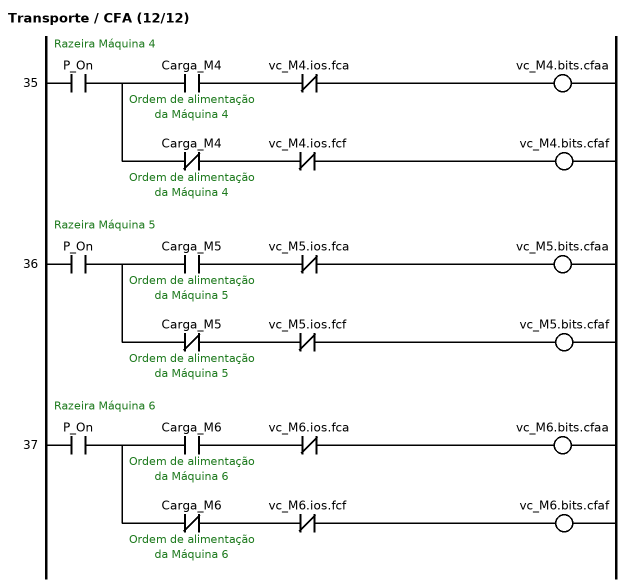
; [picture p24: Transporte / CFA, rungs 35-37]
; rung 35: Razeira Máquina 4
LD P_On
OUT TR0
AND Carga_M4  ; Ordem de alimentação da Máquina 4
ANDNOT vc_M4.ios.fca
OUT vc_M4.bits.cfaa
LD TR0
ANDNOT Carga_M4  ; Ordem de alimentação da Máquina 4
ANDNOT vc_M4.ios.fcf
OUT vc_M4.bits.cfaf
; rung 36: Razeira Máquina 5
LD P_On
OUT TR0
AND Carga_M5  ; Ordem de alimentação da Máquina 5
ANDNOT vc_M5.ios.fca
OUT vc_M5.bits.cfaa
LD TR0
ANDNOT Carga_M5  ; Ordem de alimentação da Máquina 5
ANDNOT vc_M5.ios.fcf
OUT vc_M5.bits.cfaf
; rung 37: Razeira Máquina 6
LD P_On
OUT TR0
AND Carga_M6  ; Ordem de alimentação da Máquina 6
ANDNOT vc_M6.ios.fca
OUT vc_M6.bits.cfaa
LD TR0
ANDNOT Carga_M6  ; Ordem de alimentação da Máquina 6
ANDNOT vc_M6.ios.fcf
OUT vc_M6.bits.cfaf

### Section FCOMUNICACAO

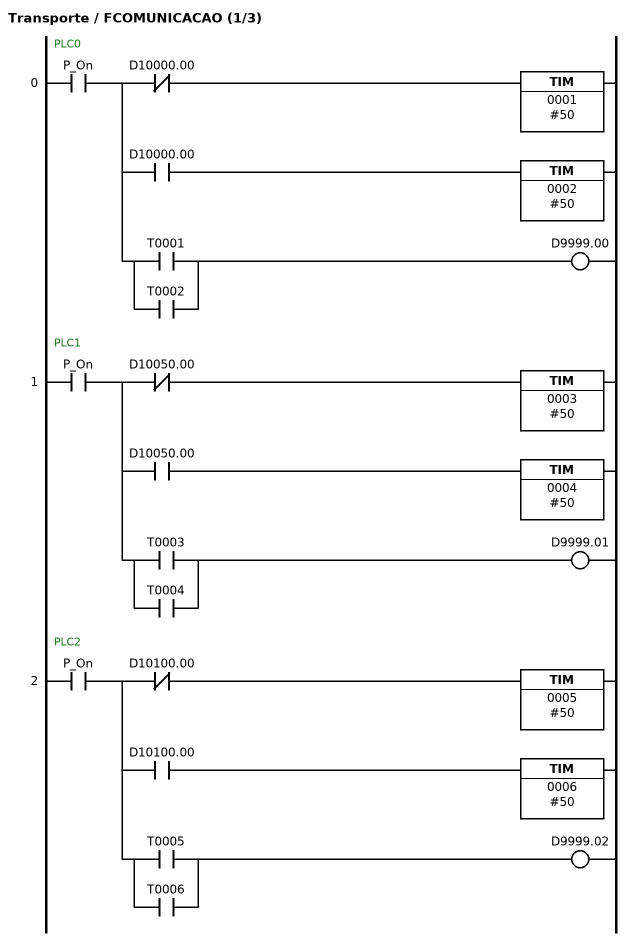
; rung 0: PLC0
LD P_On
OUT TR0
ANDNOT D10000.00
TIM 0001 #50
LD TR0
AND D10000.00
TIM 0002 #50
LD TR0
LD T0001
OR T0002
ANDLD
OUT D9999.00
; rung 1: PLC1
LD P_On
OUT TR0
ANDNOT D10050.00
TIM 0003 #50
LD TR0
AND D10050.00
TIM 0004 #50
LD TR0
LD T0003
OR T0004
ANDLD
OUT D9999.01
; rung 2: PLC2
LD P_On
OUT TR0
ANDNOT D10100.00
TIM 0005 #50
LD TR0
AND D10100.00
TIM 0006 #50
LD TR0
LD T0005
OR T0006
ANDLD
OUT D9999.02

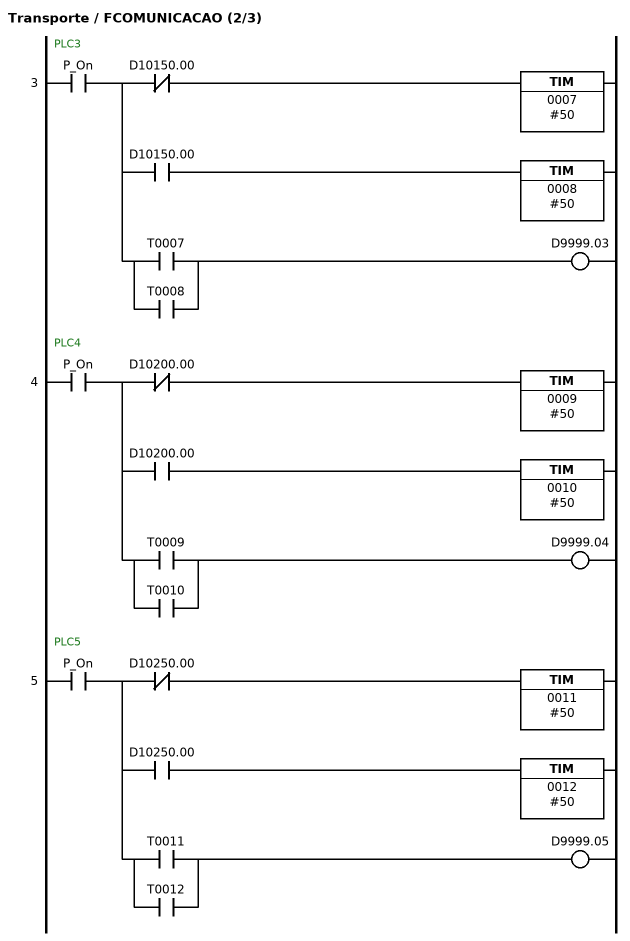
; rung 3: PLC3
LD P_On
OUT TR0
ANDNOT D10150.00
TIM 0007 #50
LD TR0
AND D10150.00
TIM 0008 #50
LD TR0
LD T0007
OR T0008
ANDLD
OUT D9999.03
; rung 4: PLC4
LD P_On
OUT TR0
ANDNOT D10200.00
TIM 0009 #50
LD TR0
AND D10200.00
TIM 0010 #50
LD TR0
LD T0009
OR T0010
ANDLD
OUT D9999.04
; rung 5: PLC5
LD P_On
OUT TR0
ANDNOT D10250.00
TIM 0011 #50
LD TR0
AND D10250.00
TIM 0012 #50
LD TR0
LD T0011
OR T0012
ANDLD
OUT D9999.05

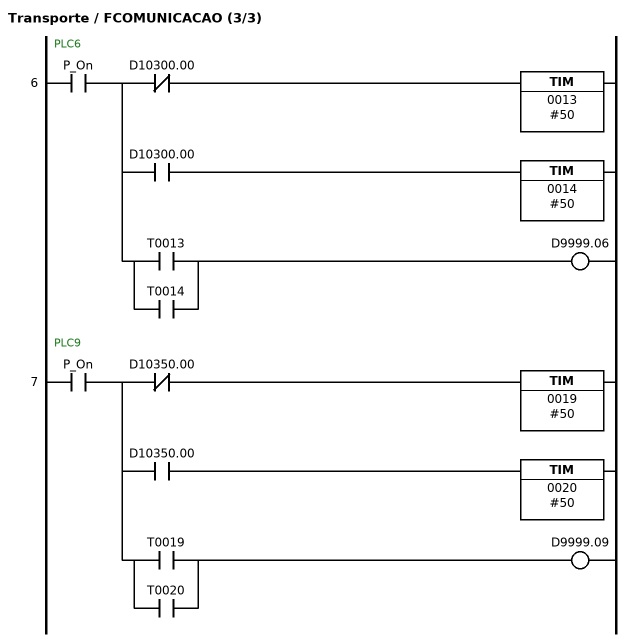
; rung 6: PLC6
LD P_On
OUT TR0
ANDNOT D10300.00
TIM 0013 #50
LD TR0
AND D10300.00
TIM 0014 #50
LD TR0
LD T0013
OR T0014
ANDLD
OUT D9999.06
; rung 7: PLC9
LD P_On
OUT TR0
ANDNOT D10350.00
TIM 0019 #50
LD TR0
AND D10350.00
TIM 0020 #50
LD TR0
LD T0019
OR T0020
ANDLD
OUT D9999.09

### Section COMUNICACAO

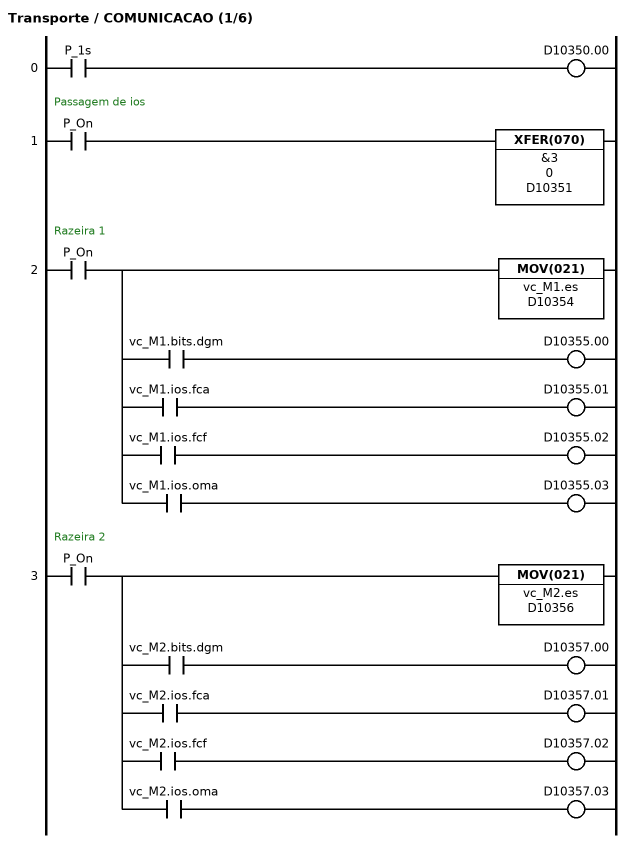
; rung 0
LD P_1s
OUT D10350.00
; rung 1: Passagem de ios
LD P_On
XFER(070) &3 0 D10351
; rung 2: Razeira 1
LD P_On
OUT TR0
MOV(021) vc_M1.es D10354
AND vc_M1.bits.dgm
OUT D10355.00
LD TR0
AND vc_M1.ios.fca
OUT D10355.01
LD TR0
AND vc_M1.ios.fcf
OUT D10355.02
LD TR0
AND vc_M1.ios.oma
OUT D10355.03
; rung 3: Razeira 2
LD P_On
OUT TR0
MOV(021) vc_M2.es D10356
AND vc_M2.bits.dgm
OUT D10357.00
LD TR0
AND vc_M2.ios.fca
OUT D10357.01
LD TR0
AND vc_M2.ios.fcf
OUT D10357.02
LD TR0
AND vc_M2.ios.oma
OUT D10357.03

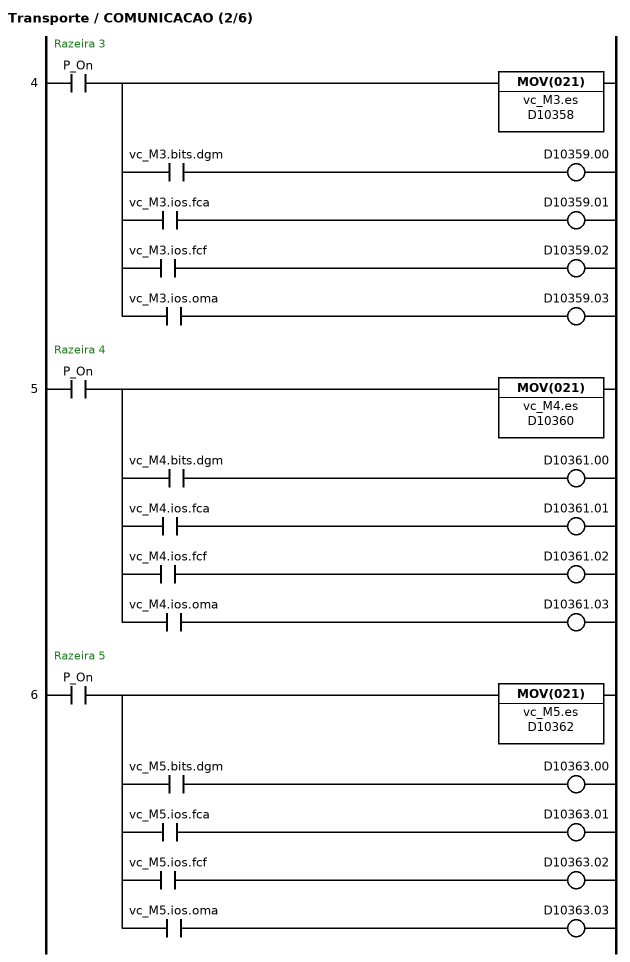
; rung 4: Razeira 3
LD P_On
OUT TR0
MOV(021) vc_M3.es D10358
AND vc_M3.bits.dgm
OUT D10359.00
LD TR0
AND vc_M3.ios.fca
OUT D10359.01
LD TR0
AND vc_M3.ios.fcf
OUT D10359.02
LD TR0
AND vc_M3.ios.oma
OUT D10359.03
; rung 5: Razeira 4
LD P_On
OUT TR0
MOV(021) vc_M4.es D10360
AND vc_M4.bits.dgm
OUT D10361.00
LD TR0
AND vc_M4.ios.fca
OUT D10361.01
LD TR0
AND vc_M4.ios.fcf
OUT D10361.02
LD TR0
AND vc_M4.ios.oma
OUT D10361.03
; rung 6: Razeira 5
LD P_On
OUT TR0
MOV(021) vc_M5.es D10362
AND vc_M5.bits.dgm
OUT D10363.00
LD TR0
AND vc_M5.ios.fca
OUT D10363.01
LD TR0
AND vc_M5.ios.fcf
OUT D10363.02
LD TR0
AND vc_M5.ios.oma
OUT D10363.03

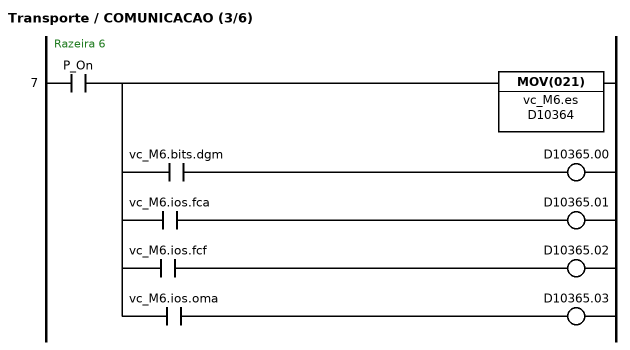
; rung 7: Razeira 6
LD P_On
OUT TR0
MOV(021) vc_M6.es D10364
AND vc_M6.bits.dgm
OUT D10365.00
LD TR0
AND vc_M6.ios.fca
OUT D10365.01
LD TR0
AND vc_M6.ios.fcf
OUT D10365.02
LD TR0
AND vc_M6.ios.oma
OUT D10365.03

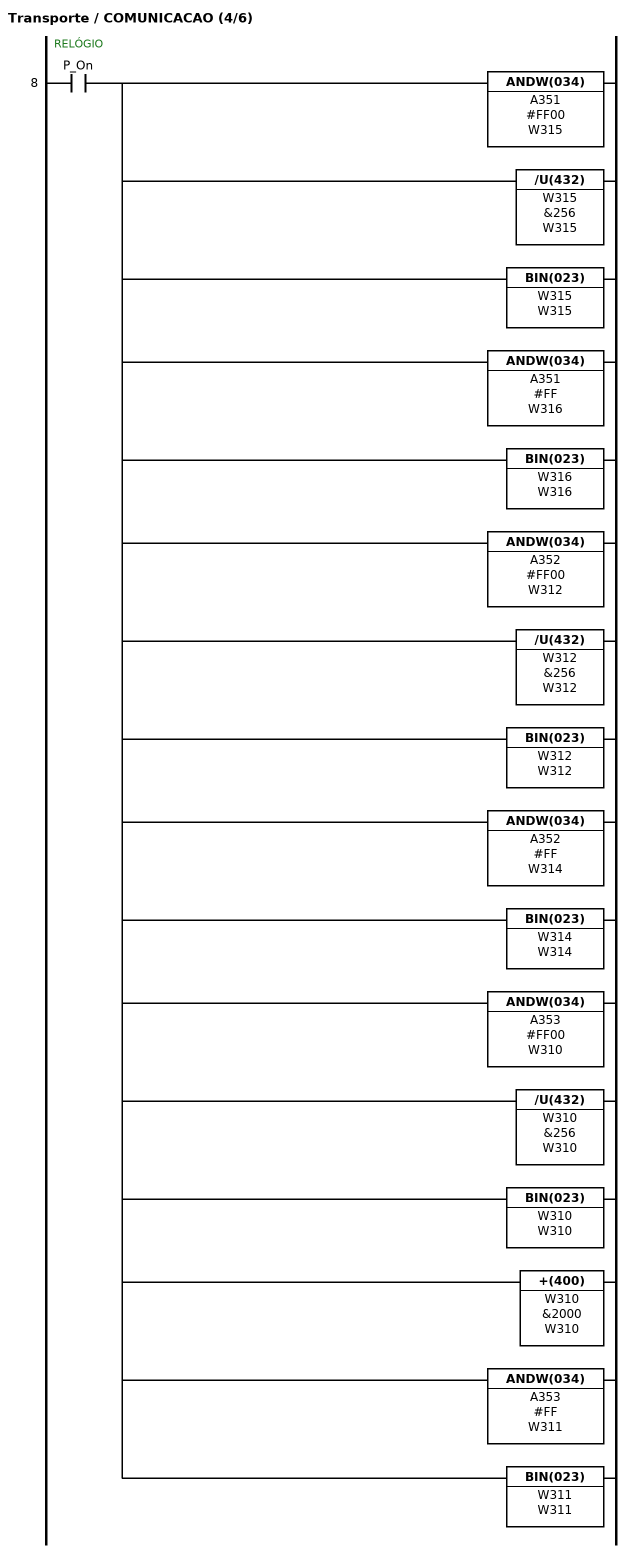
; rung 8: RELÓGIO
LD P_On
ANDW(034) A351 #FF00 W315
/U(432) W315 &256 W315
BIN(023) W315 W315
ANDW(034) A351 #FF W316
BIN(023) W316 W316
ANDW(034) A352 #FF00 W312
/U(432) W312 &256 W312
BIN(023) W312 W312
ANDW(034) A352 #FF W314
BIN(023) W314 W314
ANDW(034) A353 #FF00 W310
/U(432) W310 &256 W310
BIN(023) W310 W310
+(400) W310 &2000 W310
ANDW(034) A353 #FF W311
BIN(023) W311 W311

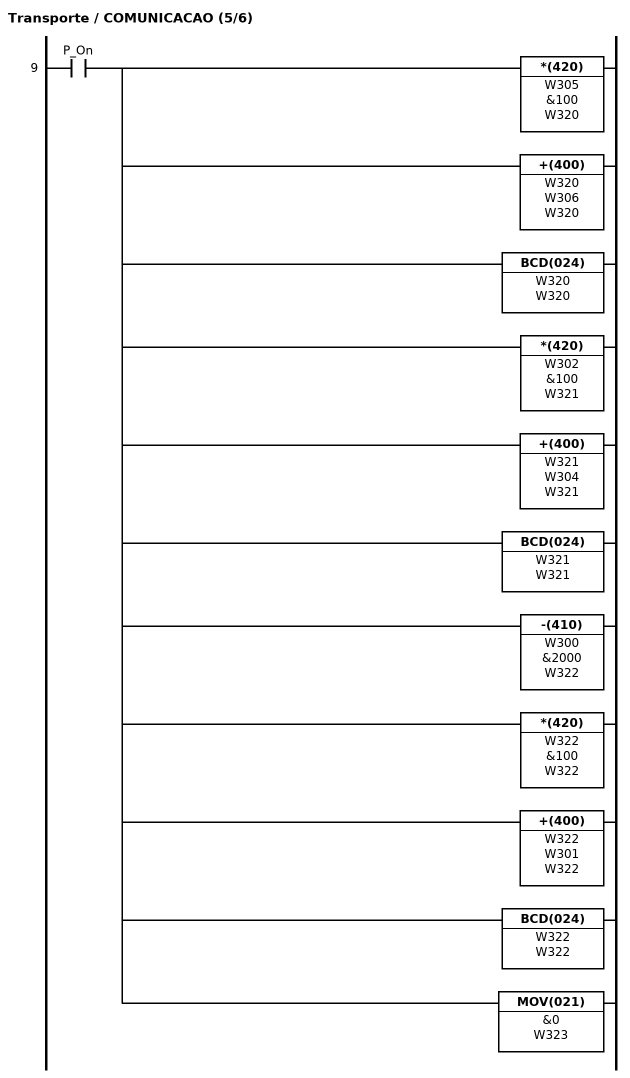
; rung 9
LD P_On
*(420) W305 &100 W320
+(400) W320 W306 W320
BCD(024) W320 W320
*(420) W302 &100 W321
+(400) W321 W304 W321
BCD(024) W321 W321
-(410) W300 &2000 W322
*(420) W322 &100 W322
+(400) W322 W301 W322
BCD(024) W322 W322
MOV(021) &0 W323

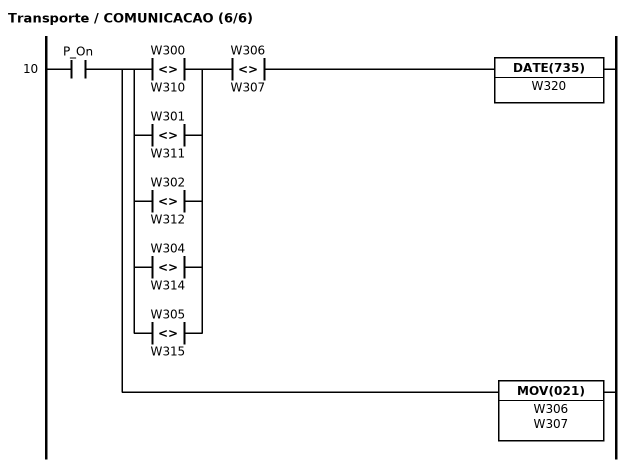
; rung 10
LD P_On
OUT TR0
LD<>(305) W300 W310
OR<>(305) W301 W311
OR<>(305) W302 W312
OR<>(305) W304 W314
OR<>(305) W305 W315
ANDLD
AND<>(305) W306 W307
DATE(735) W320
LD TR0
MOV(021) W306 W307

### Section Comm_MasterPLC

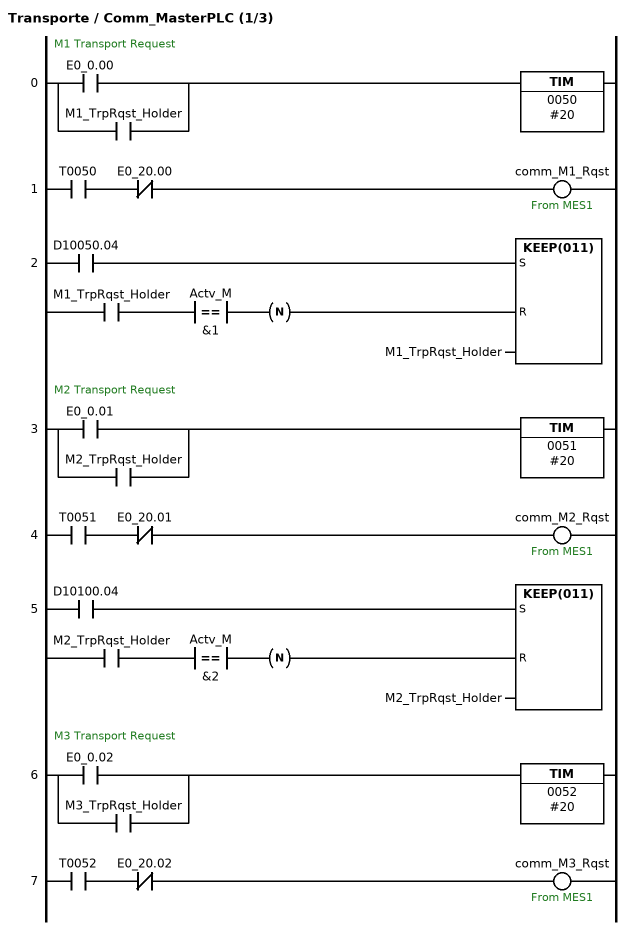
; rung 0: M1 Transport Request
LD E0_0.00
OR M1_TrpRqst_Holder
TIM 0050 #20
; rung 1
LD T0050
ANDNOT E0_20.00
OUT comm_M1_Rqst  ; From MES1
; rung 2
LD D10050.04
LD M1_TrpRqst_Holder
AND=(300) Actv_M &1
DOWN(522)
KEEP(011) M1_TrpRqst_Holder
; rung 3: M2 Transport Request
LD E0_0.01
OR M2_TrpRqst_Holder
TIM 0051 #20
; rung 4
LD T0051
ANDNOT E0_20.01
OUT comm_M2_Rqst  ; From MES1
; rung 5
LD D10100.04
LD M2_TrpRqst_Holder
AND=(300) Actv_M &2
DOWN(522)
KEEP(011) M2_TrpRqst_Holder
; rung 6: M3 Transport Request
LD E0_0.02
OR M3_TrpRqst_Holder
TIM 0052 #20
; rung 7
LD T0052
ANDNOT E0_20.02
OUT comm_M3_Rqst  ; From MES1

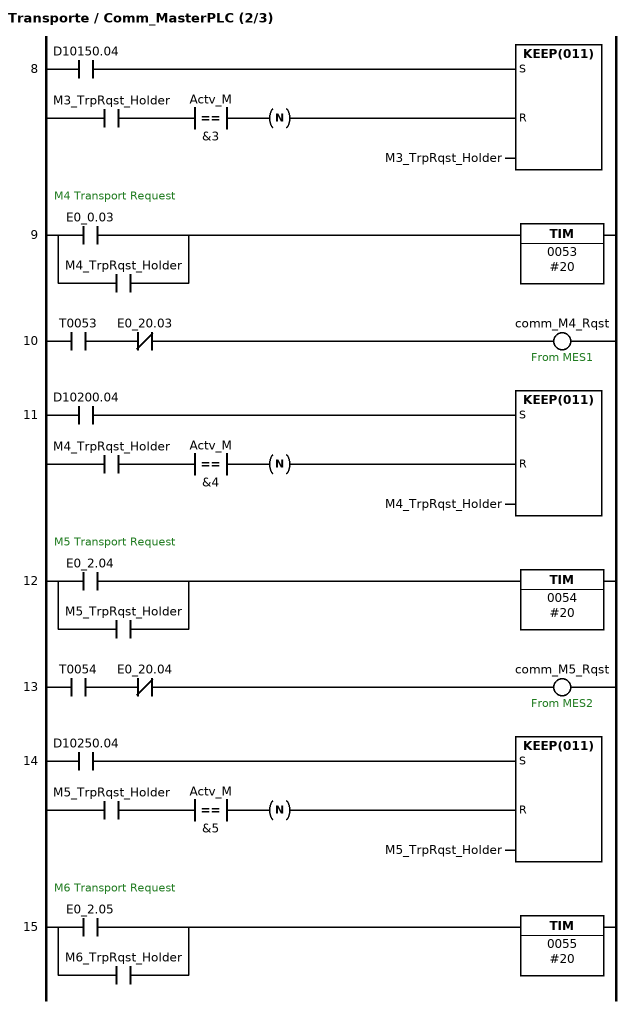
; rung 8
LD D10150.04
LD M3_TrpRqst_Holder
AND=(300) Actv_M &3
DOWN(522)
KEEP(011) M3_TrpRqst_Holder
; rung 9: M4 Transport Request
LD E0_0.03
OR M4_TrpRqst_Holder
TIM 0053 #20
; rung 10
LD T0053
ANDNOT E0_20.03
OUT comm_M4_Rqst  ; From MES1
; rung 11
LD D10200.04
LD M4_TrpRqst_Holder
AND=(300) Actv_M &4
DOWN(522)
KEEP(011) M4_TrpRqst_Holder
; rung 12: M5 Transport Request
LD E0_2.04
OR M5_TrpRqst_Holder
TIM 0054 #20
; rung 13
LD T0054
ANDNOT E0_20.04
OUT comm_M5_Rqst  ; From MES2
; rung 14
LD D10250.04
LD M5_TrpRqst_Holder
AND=(300) Actv_M &5
DOWN(522)
KEEP(011) M5_TrpRqst_Holder
; rung 15: M6 Transport Request
LD E0_2.05
OR M6_TrpRqst_Holder
TIM 0055 #20

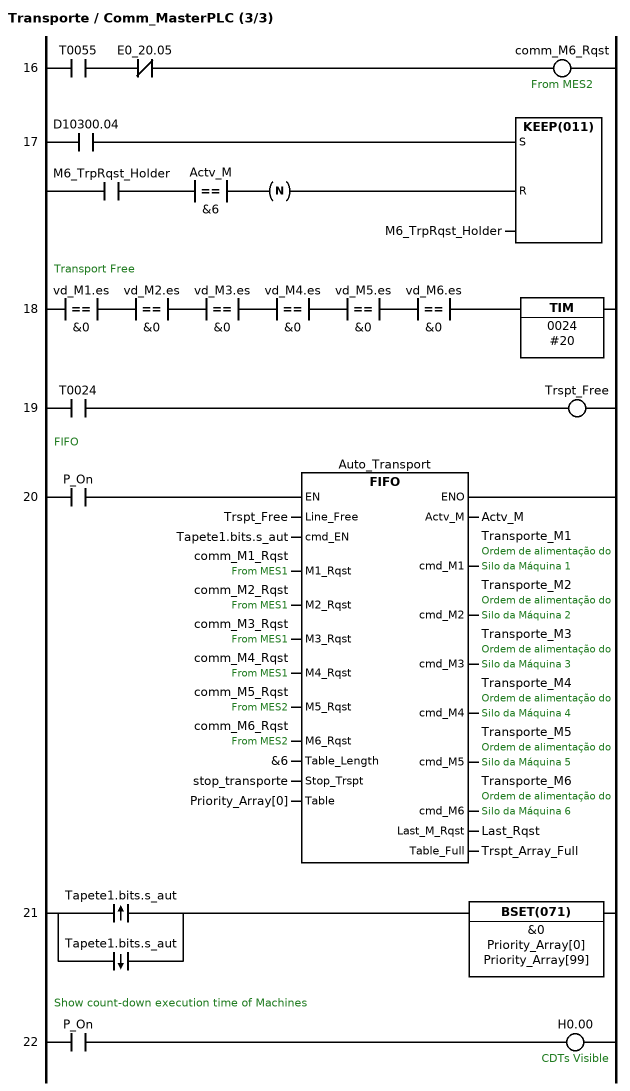
; rung 16
LD T0055
ANDNOT E0_20.05
OUT comm_M6_Rqst  ; From MES2
; rung 17
LD D10300.04
LD M6_TrpRqst_Holder
AND=(300) Actv_M &6
DOWN(522)
KEEP(011) M6_TrpRqst_Holder
; rung 18: Transport Free
LD=(300) vd_M1.es &0
AND=(300) vd_M2.es &0
AND=(300) vd_M3.es &0
AND=(300) vd_M4.es &0
AND=(300) vd_M5.es &0
AND=(300) vd_M6.es &0
TIM 0024 #20
; rung 19
LD T0024
OUT Trspt_Free
; rung 20: FIFO
LD P_On
CALL Auto_Transport : FIFO (Line_Free := Trspt_Free, cmd_EN := Tapete1.bits.s_aut, M1_Rqst := comm_M1_Rqst, M2_Rqst := comm_M2_Rqst, M3_Rqst := comm_M3_Rqst, M4_Rqst := comm_M4_Rqst, M5_Rqst := comm_M5_Rqst, M6_Rqst := comm_M6_Rqst, Table_Length := &6, Stop_Trspt := stop_transporte, Table := Priority_Array[0], Actv_M => Actv_M, cmd_M1 => Transporte_M1, cmd_M2 => Transporte_M2, cmd_M3 => Transporte_M3, cmd_M4 => Transporte_M4, cmd_M5 => Transporte_M5, cmd_M6 => Transporte_M6, Last_M_Rqst => Last_Rqst, Table_Full => Trspt_Array_Full)  ; From MES1, From MES2, Ordem de alimentação do Silo da Máquina 1, Ordem de alimentação do Silo da Máquina 2, Ordem de alimentação do Silo da Máquina 3, Ordem de alimentação do Silo da Máquina 4, Ordem de alimentação do Silo da Máquina 5, Ordem de alimentação do Silo da Máquina 6
; rung 21
@LD Tapete1.bits.s_aut
%OR Tapete1.bits.s_aut
BSET(071) &0 Priority_Array[0] Priority_Array[99]
; rung 22: Show count-down execution time of Machines
LD P_On
OUT H0.00  ; CDTs Visible

### Section END
; rung 0
END(001)

## Function block Array_Analysis
VAR_INPUT
  First_index : INT;
  Last_index : INT;
END_VAR
VAR_OUTPUT
  Empty_Index : INT;
  Ary_Full : BOOL;
  Last_Member : INT;
END_VAR
VAR_IN_OUT
  Ary : ARRAY[0..99] OF INT;
END_VAR
VAR
  itr : INT;
  Loop_Stop : BOOL;
END_VAR
Loop_Stop := FALSE;
Last_Member := 0;

FOR itr := First_index TO Last_index DO
IF Ary[itr]=0 AND  NOT Loop_Stop THEN
	Empty_Index := itr;
	Loop_Stop := TRUE;
END_IF;

IF Ary[itr]<>0  THEN
	Last_Member := Ary[itr];
END_IF;
END_FOR;

IF Ary[Last_index] <> 0 THEN
	Ary_Full := TRUE;
	Empty_Index := -1;
ELSE
	Ary_Full := FALSE;
END_IF;

## Function block Array_Search
VAR_INPUT
  Member : INT;
  First_index : INT;
  Last_index : INT;
END_VAR
VAR_OUTPUT
  Indx : INT;
END_VAR
VAR_IN_OUT
  Ary : ARRAY[0..99] OF INT;
END_VAR
VAR
  Loop_Stop : BOOL;
  itr : INT;
END_VAR
Loop_Stop := FALSE;
Indx :=  -1;

FOR itr := First_index TO Last_index DO
IF Ary[itr]=Member AND  NOT Loop_Stop THEN
	Indx :=  itr;
	Loop_Stop := TRUE;
END_IF;
END_FOR;

## Function block fb_eq_motor
; FUNÇÃO MOTOR - Controlo de uma maquina tipo motor.
VAR_IN_OUT
  mot : s_equip;  (* Dados do motor *)
END_VAR
VAR
  tm01 : TIMER;
END_VAR

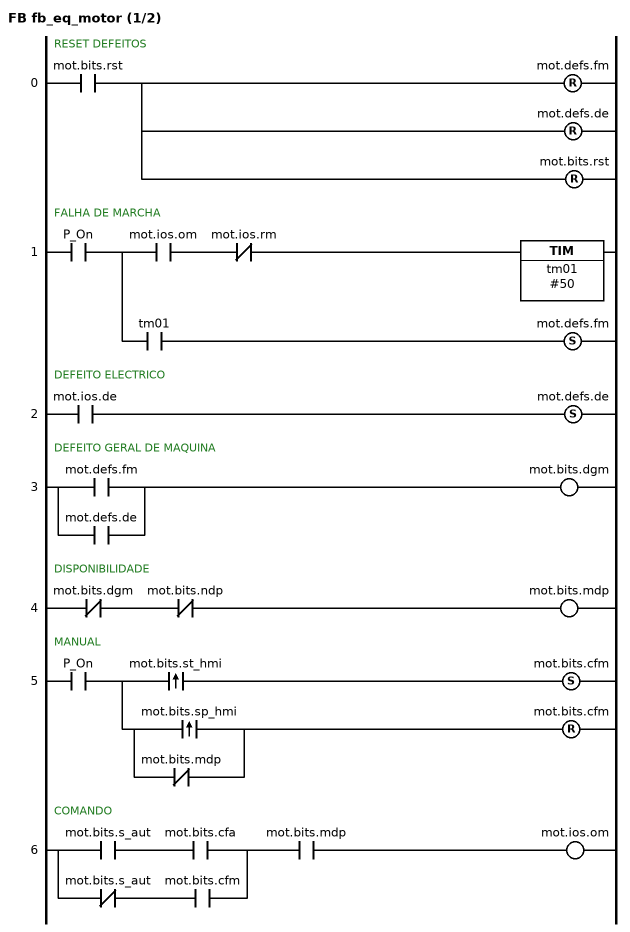
; rung 0: RESET DEFEITOS
LD mot.bits.rst
RSET mot.defs.fm
RSET mot.defs.de
RSET mot.bits.rst
; rung 1: FALHA DE MARCHA
LD P_On
OUT TR0
AND mot.ios.om
ANDNOT mot.ios.rm
TIM tm01 #50
LD TR0
AND tm01
SET mot.defs.fm
; rung 2: DEFEITO ELECTRICO
LD mot.ios.de
SET mot.defs.de
; rung 3: DEFEITO GERAL DE MAQUINA
LD mot.defs.fm
OR mot.defs.de
OUT mot.bits.dgm
; rung 4: DISPONIBILIDADE
LDNOT mot.bits.dgm
ANDNOT mot.bits.ndp
OUT mot.bits.mdp
; rung 5: MANUAL
LD P_On
OUT TR0
@AND mot.bits.st_hmi
SET mot.bits.cfm
LD TR0
@LD mot.bits.sp_hmi
ORNOT mot.bits.mdp
ANDLD
RSET mot.bits.cfm
; rung 6: COMANDO
LD mot.bits.s_aut
AND mot.bits.cfa
LDNOT mot.bits.s_aut
AND mot.bits.cfm
ORLD
AND mot.bits.mdp
OUT mot.ios.om

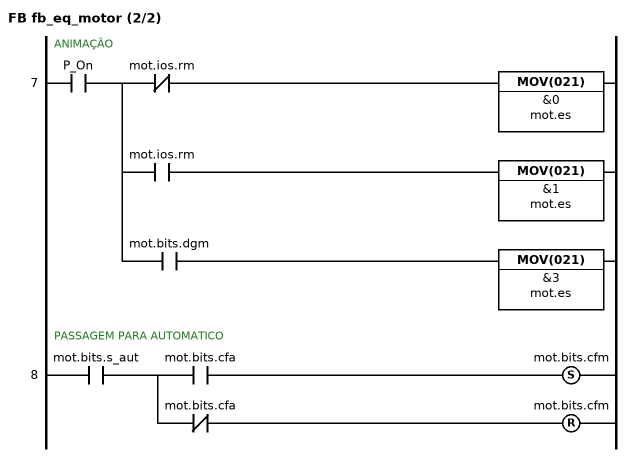
; rung 7: ANIMAÇÃO
LD P_On
OUT TR0
ANDNOT mot.ios.rm
MOV(021) &0 mot.es
LD TR0
AND mot.ios.rm
MOV(021) &1 mot.es
LD TR0
AND mot.bits.dgm
MOV(021) &3 mot.es
; rung 8: PASSAGEM PARA AUTOMATICO
LD mot.bits.s_aut
OUT TR0
AND mot.bits.cfa
SET mot.bits.cfm
LD TR0
ANDNOT mot.bits.cfa
RSET mot.bits.cfm

## Function block fb_eq_valvula
; FUNÇÃO VALVULA - Controlo de uma maquina tipo valvula.
VAR_IN_OUT
  valv : s_equip;  (* Dados da valvula *)
END_VAR
VAR
  tm01 : TIMER;
  tm02 : TIMER;
END_VAR

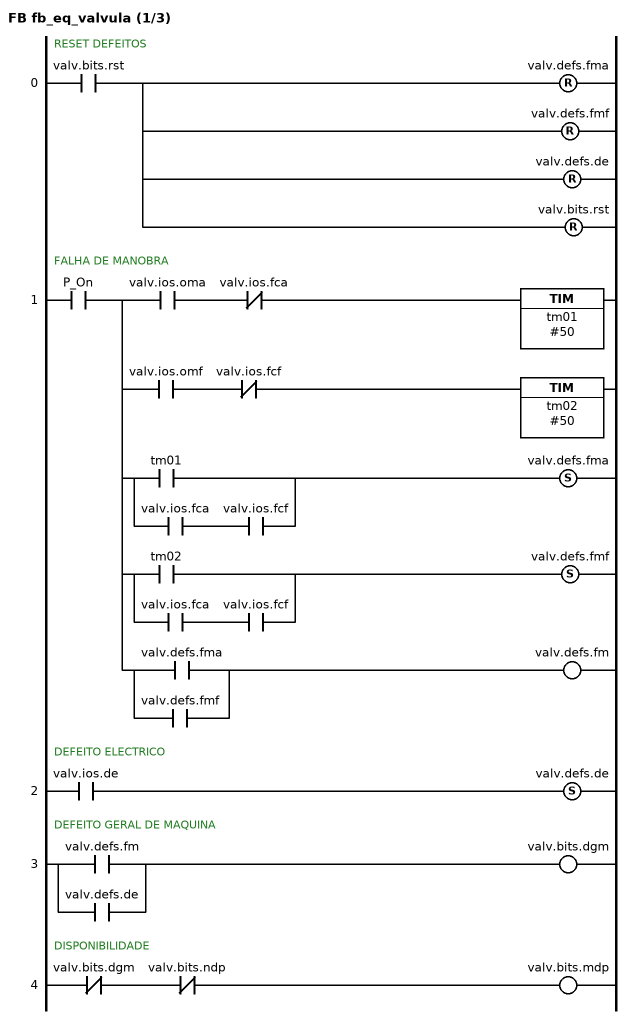
; rung 0: RESET DEFEITOS
LD valv.bits.rst
RSET valv.defs.fma
RSET valv.defs.fmf
RSET valv.defs.de
RSET valv.bits.rst
; rung 1: FALHA DE MANOBRA
LD P_On
OUT TR0
AND valv.ios.oma
ANDNOT valv.ios.fca
TIM tm01 #50
LD TR0
AND valv.ios.omf
ANDNOT valv.ios.fcf
TIM tm02 #50
LD TR0
LD tm01
LD valv.ios.fca
AND valv.ios.fcf
ORLD
ANDLD
SET valv.defs.fma
LD TR0
LD tm02
LD valv.ios.fca
AND valv.ios.fcf
ORLD
ANDLD
SET valv.defs.fmf
LD TR0
LD valv.defs.fma
OR valv.defs.fmf
ANDLD
OUT valv.defs.fm
; rung 2: DEFEITO ELECTRICO
LD valv.ios.de
SET valv.defs.de
; rung 3: DEFEITO GERAL DE MAQUINA
LD valv.defs.fm
OR valv.defs.de
OUT valv.bits.dgm
; rung 4: DISPONIBILIDADE
LDNOT valv.bits.dgm
ANDNOT valv.bits.ndp
OUT valv.bits.mdp

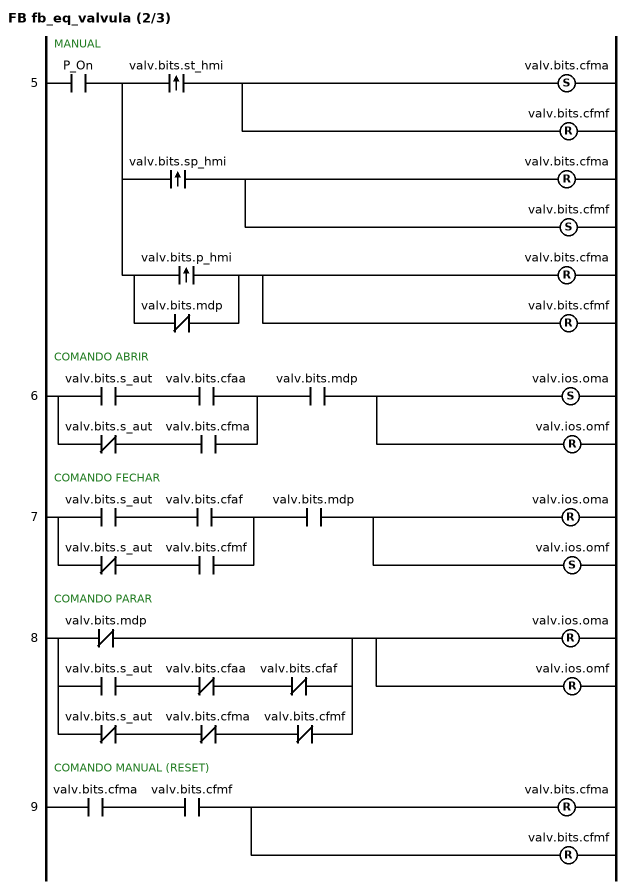
; rung 5: MANUAL
LD P_On
OUT TR0
@AND valv.bits.st_hmi
SET valv.bits.cfma
RSET valv.bits.cfmf
LD TR0
@AND valv.bits.sp_hmi
RSET valv.bits.cfma
SET valv.bits.cfmf
LD TR0
@LD valv.bits.p_hmi
ORNOT valv.bits.mdp
ANDLD
RSET valv.bits.cfma
RSET valv.bits.cfmf
; rung 6: COMANDO ABRIR
LD valv.bits.s_aut
AND valv.bits.cfaa
LDNOT valv.bits.s_aut
AND valv.bits.cfma
ORLD
AND valv.bits.mdp
SET valv.ios.oma
RSET valv.ios.omf
; rung 7: COMANDO FECHAR
LD valv.bits.s_aut
AND valv.bits.cfaf
LDNOT valv.bits.s_aut
AND valv.bits.cfmf
ORLD
AND valv.bits.mdp
RSET valv.ios.oma
SET valv.ios.omf
; rung 8: COMANDO PARAR
LDNOT valv.bits.mdp
LD valv.bits.s_aut
ANDNOT valv.bits.cfaa
ANDNOT valv.bits.cfaf
ORLD
LDNOT valv.bits.s_aut
ANDNOT valv.bits.cfma
ANDNOT valv.bits.cfmf
ORLD
RSET valv.ios.oma
RSET valv.ios.omf
; rung 9: COMANDO MANUAL (RESET)
LD valv.bits.cfma
AND valv.bits.cfmf
RSET valv.bits.cfma
RSET valv.bits.cfmf

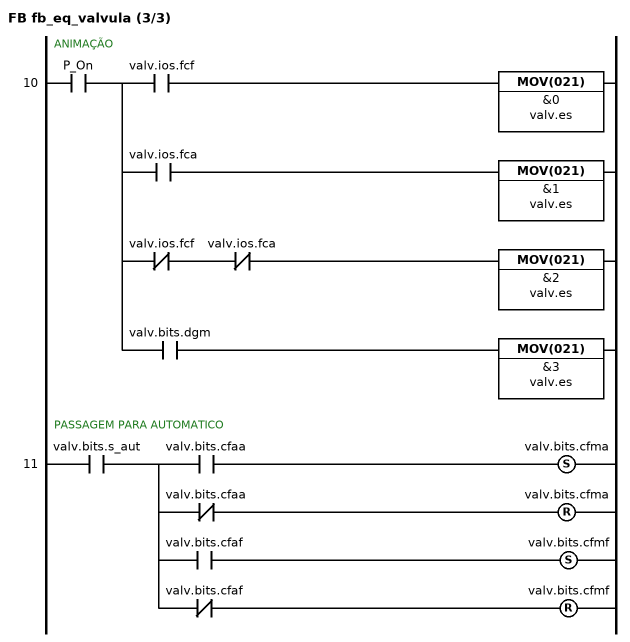
; rung 10: ANIMAÇÃO
LD P_On
OUT TR0
AND valv.ios.fcf
MOV(021) &0 valv.es
LD TR0
AND valv.ios.fca
MOV(021) &1 valv.es
LD TR0
ANDNOT valv.ios.fcf
ANDNOT valv.ios.fca
MOV(021) &2 valv.es
LD TR0
AND valv.bits.dgm
MOV(021) &3 valv.es
; rung 11: PASSAGEM PARA AUTOMATICO
LD valv.bits.s_aut
OUT TR0
AND valv.bits.cfaa
SET valv.bits.cfma
LD TR0
ANDNOT valv.bits.cfaa
RSET valv.bits.cfma
LD TR0
AND valv.bits.cfaf
SET valv.bits.cfmf
LD TR0
ANDNOT valv.bits.cfaf
RSET valv.bits.cfmf

## Function block FIFO
; This function finds the least significant position of a arry. / The seeking area can be limited by firsr arry (FstAry) and last Array (LstAry) which are the inputs of function block.
VAR_INPUT
  Line_Free : BOOL;
  cmd_EN : BOOL;
  M1_Rqst : BOOL;
  M2_Rqst : BOOL;
  M3_Rqst : BOOL;
  M4_Rqst : BOOL;
  M5_Rqst : BOOL;
  M6_Rqst : BOOL;
  Table_Length : INT;
  Stop_Trspt : BOOL;
END_VAR
VAR_OUTPUT
  Actv_M : INT;
  cmd_M1 : BOOL;
  cmd_M2 : BOOL;
  cmd_M3 : BOOL;
  cmd_M4 : BOOL;
  cmd_M5 : BOOL;
  cmd_M6 : BOOL;
  Last_M_Rqst : INT;
  Table_Full : BOOL;
END_VAR
VAR_IN_OUT
  Table : ARRAY[0..99] OF INT;
END_VAR
VAR
  M_Rqst_tmp : INT;
  Empty_Position : INT;
  Shift_Table : Shift_Ary;
  Tabel_LstIndx : INT;
  Table_Analysis : Array_Analysis;
  M1_Position : INT;
  Cancel_Rqst_Indx : INT;
  M2_Position : INT;
  M3_Position : INT;
  M4_Position : INT;
  M5_Position : INT;
  M6_Position : INT;
  Search_M1 : Array_Search;
  Search_M2 : Array_Search;
  Search_M3 : Array_Search;
  Search_M4 : Array_Search;
  Search_M5 : Array_Search;
  Search_M6 : Array_Search;
  Cancel_Rqst : Shift_Ary;
  Cancel_Rqst_cmd : BOOL;
  Neg_one : INT;
  cmd_Shift : BOOL;
END_VAR

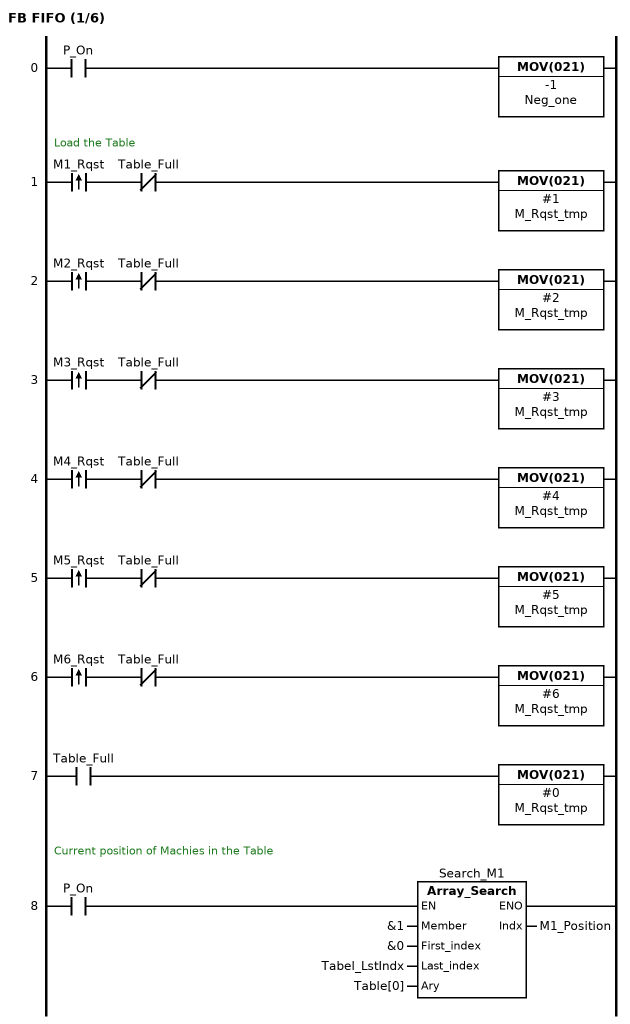
; rung 0
LD P_On
MOV(021) -1 Neg_one
; rung 1: Load the Table
@LD M1_Rqst
ANDNOT Table_Full
MOV(021) #1 M_Rqst_tmp
; rung 2
@LD M2_Rqst
ANDNOT Table_Full
MOV(021) #2 M_Rqst_tmp
; rung 3
@LD M3_Rqst
ANDNOT Table_Full
MOV(021) #3 M_Rqst_tmp
; rung 4
@LD M4_Rqst
ANDNOT Table_Full
MOV(021) #4 M_Rqst_tmp
; rung 5
@LD M5_Rqst
ANDNOT Table_Full
MOV(021) #5 M_Rqst_tmp
; rung 6
@LD M6_Rqst
ANDNOT Table_Full
MOV(021) #6 M_Rqst_tmp
; rung 7
LD Table_Full
MOV(021) #0 M_Rqst_tmp
; rung 8: Current position of Machies in the Table
LD P_On
CALL Search_M1 : Array_Search (Member := &1, First_index := &0, Last_index := Tabel_LstIndx, Ary := Table[0], Indx => M1_Position)

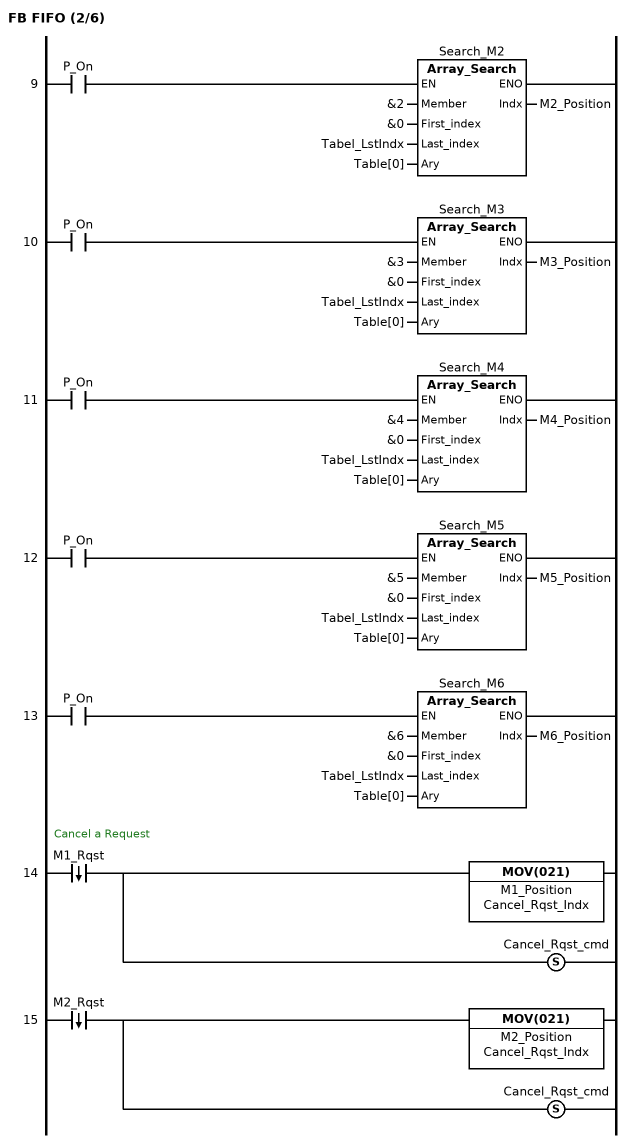
; rung 9
LD P_On
CALL Search_M2 : Array_Search (Member := &2, First_index := &0, Last_index := Tabel_LstIndx, Ary := Table[0], Indx => M2_Position)
; rung 10
LD P_On
CALL Search_M3 : Array_Search (Member := &3, First_index := &0, Last_index := Tabel_LstIndx, Ary := Table[0], Indx => M3_Position)
; rung 11
LD P_On
CALL Search_M4 : Array_Search (Member := &4, First_index := &0, Last_index := Tabel_LstIndx, Ary := Table[0], Indx => M4_Position)
; rung 12
LD P_On
CALL Search_M5 : Array_Search (Member := &5, First_index := &0, Last_index := Tabel_LstIndx, Ary := Table[0], Indx => M5_Position)
; rung 13
LD P_On
CALL Search_M6 : Array_Search (Member := &6, First_index := &0, Last_index := Tabel_LstIndx, Ary := Table[0], Indx => M6_Position)
; rung 14: Cancel a Request
%LD M1_Rqst
MOV(021) M1_Position Cancel_Rqst_Indx
SET Cancel_Rqst_cmd
; rung 15
%LD M2_Rqst
MOV(021) M2_Position Cancel_Rqst_Indx
SET Cancel_Rqst_cmd

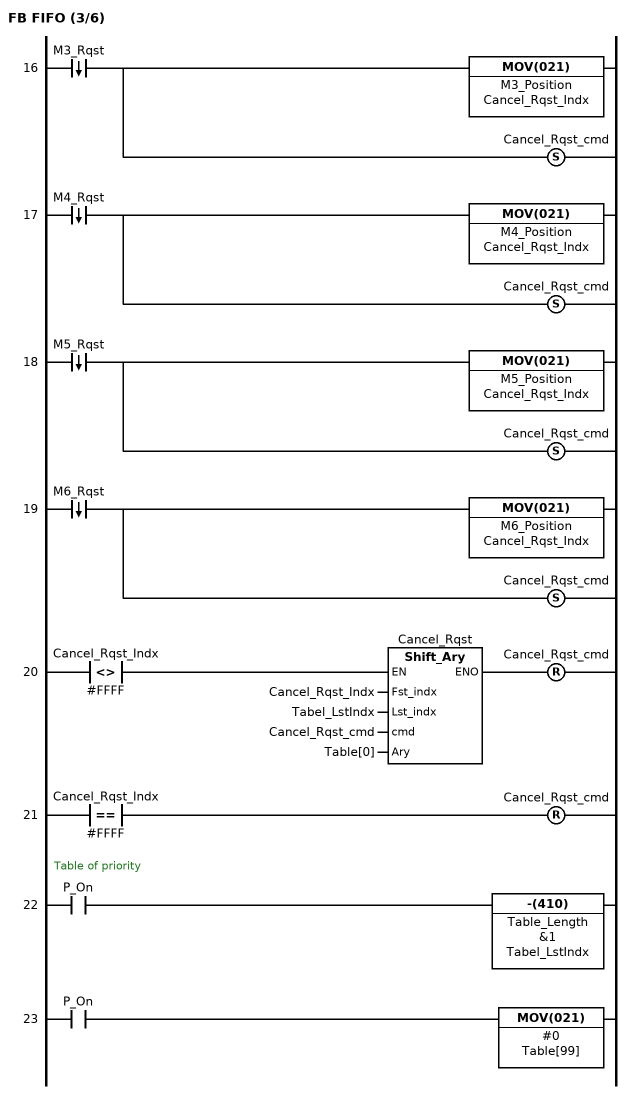
; rung 16
%LD M3_Rqst
MOV(021) M3_Position Cancel_Rqst_Indx
SET Cancel_Rqst_cmd
; rung 17
%LD M4_Rqst
MOV(021) M4_Position Cancel_Rqst_Indx
SET Cancel_Rqst_cmd
; rung 18
%LD M5_Rqst
MOV(021) M5_Position Cancel_Rqst_Indx
SET Cancel_Rqst_cmd
; rung 19
%LD M6_Rqst
MOV(021) M6_Position Cancel_Rqst_Indx
SET Cancel_Rqst_cmd
; rung 20
LD<>(305) Cancel_Rqst_Indx #FFFF
CALL Cancel_Rqst : Shift_Ary (Fst_indx := Cancel_Rqst_Indx, Lst_indx := Tabel_LstIndx, cmd := Cancel_Rqst_cmd, Ary := Table[0])
RSET Cancel_Rqst_cmd
; rung 21
LD=(300) Cancel_Rqst_Indx #FFFF
RSET Cancel_Rqst_cmd
; rung 22: Table of priority
LD P_On
-(410) Table_Length &1 Tabel_LstIndx
; rung 23
LD P_On
MOV(021) #0 Table[99]

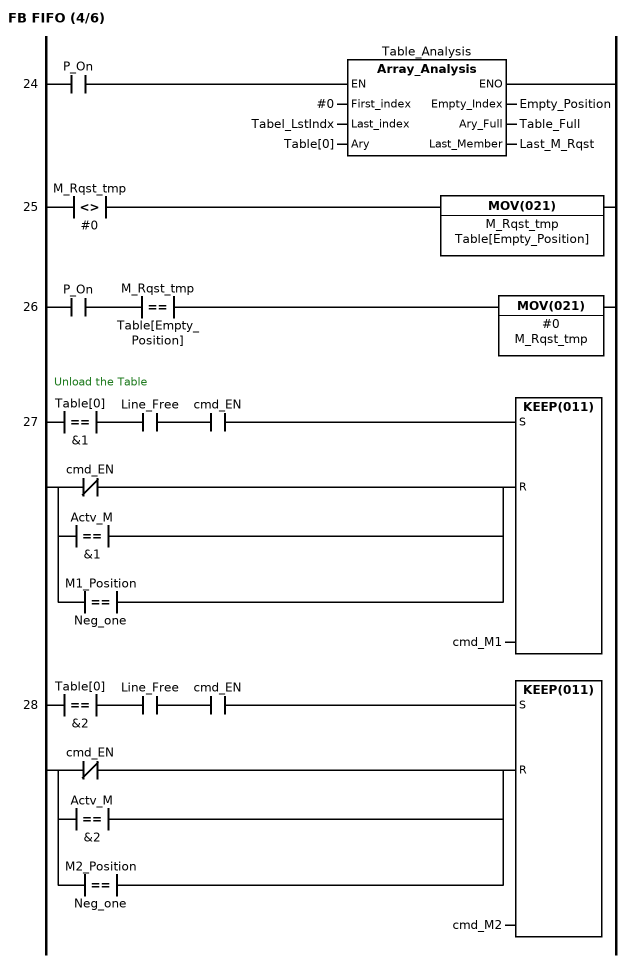
; rung 24
LD P_On
CALL Table_Analysis : Array_Analysis (First_index := #0, Last_index := Tabel_LstIndx, Ary := Table[0], Empty_Index => Empty_Position, Ary_Full => Table_Full, Last_Member => Last_M_Rqst)
; rung 25
LD<>(305) M_Rqst_tmp #0
MOV(021) M_Rqst_tmp Table[Empty_Position]
; rung 26
LD P_On
AND=(300) M_Rqst_tmp Table[Empty_Position]
MOV(021) #0 M_Rqst_tmp
; rung 27: Unload the Table
LD=(300) Table[0] &1
AND Line_Free
AND cmd_EN
LDNOT cmd_EN
OR=(300) Actv_M &1
OR=(300) M1_Position Neg_one
KEEP(011) cmd_M1
; rung 28
LD=(300) Table[0] &2
AND Line_Free
AND cmd_EN
LDNOT cmd_EN
OR=(300) Actv_M &2
OR=(300) M2_Position Neg_one
KEEP(011) cmd_M2

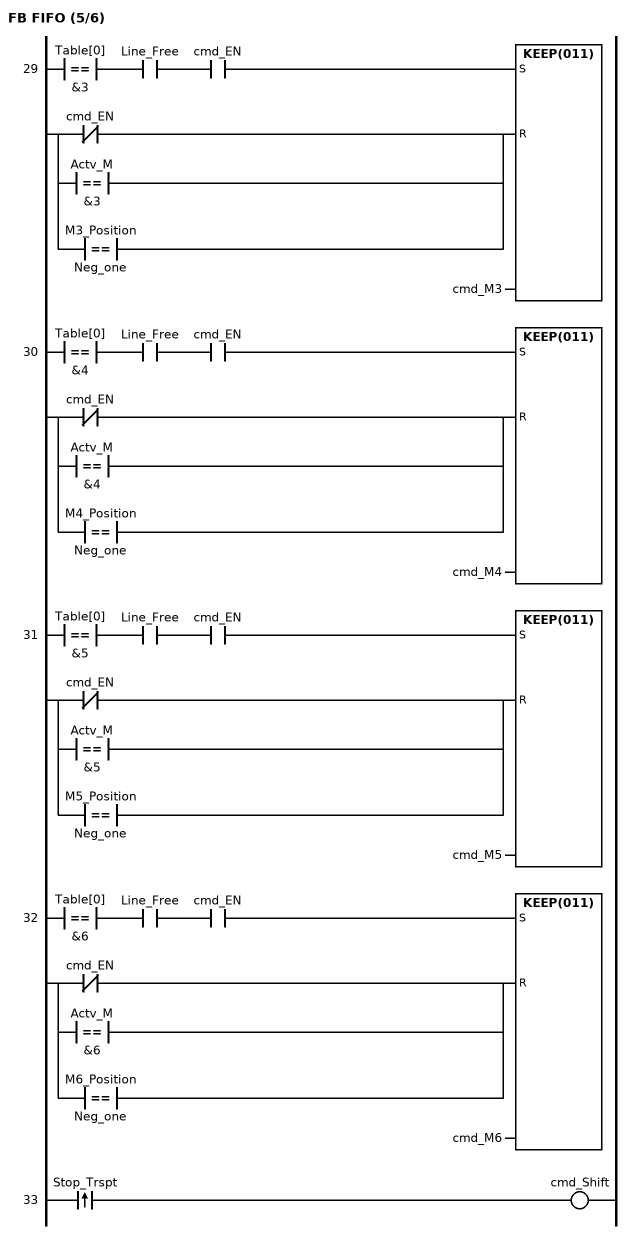
; rung 29
LD=(300) Table[0] &3
AND Line_Free
AND cmd_EN
LDNOT cmd_EN
OR=(300) Actv_M &3
OR=(300) M3_Position Neg_one
KEEP(011) cmd_M3
; rung 30
LD=(300) Table[0] &4
AND Line_Free
AND cmd_EN
LDNOT cmd_EN
OR=(300) Actv_M &4
OR=(300) M4_Position Neg_one
KEEP(011) cmd_M4
; rung 31
LD=(300) Table[0] &5
AND Line_Free
AND cmd_EN
LDNOT cmd_EN
OR=(300) Actv_M &5
OR=(300) M5_Position Neg_one
KEEP(011) cmd_M5
; rung 32
LD=(300) Table[0] &6
AND Line_Free
AND cmd_EN
LDNOT cmd_EN
OR=(300) Actv_M &6
OR=(300) M6_Position Neg_one
KEEP(011) cmd_M6
; rung 33
@LD Stop_Trspt
OUT cmd_Shift

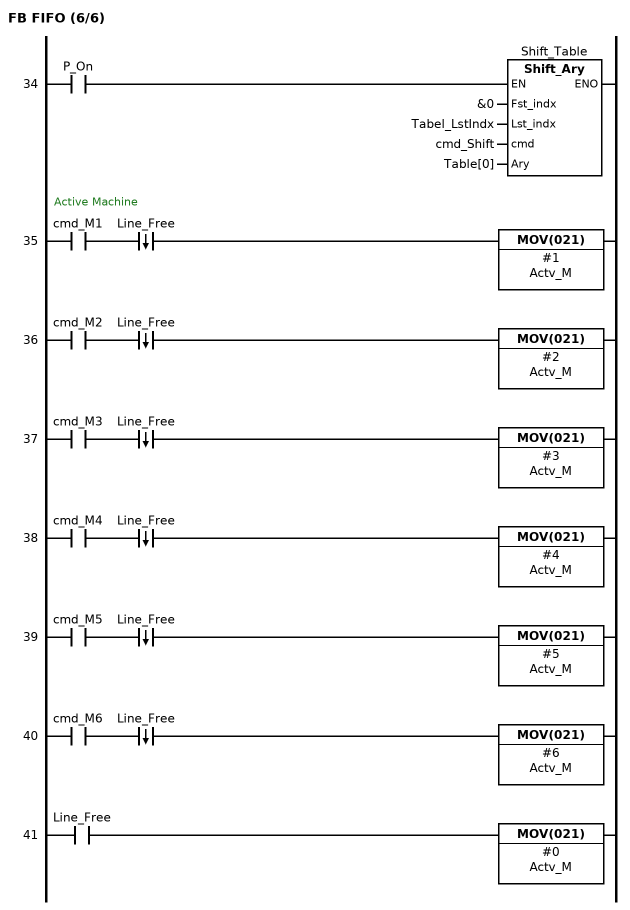
; rung 34
LD P_On
CALL Shift_Table : Shift_Ary (Fst_indx := &0, Lst_indx := Tabel_LstIndx, cmd := cmd_Shift, Ary := Table[0])
; rung 35: Active Machine
LD cmd_M1
%AND Line_Free
MOV(021) #1 Actv_M
; rung 36
LD cmd_M2
%AND Line_Free
MOV(021) #2 Actv_M
; rung 37
LD cmd_M3
%AND Line_Free
MOV(021) #3 Actv_M
; rung 38
LD cmd_M4
%AND Line_Free
MOV(021) #4 Actv_M
; rung 39
LD cmd_M5
%AND Line_Free
MOV(021) #5 Actv_M
; rung 40
LD cmd_M6
%AND Line_Free
MOV(021) #6 Actv_M
; rung 41
LD Line_Free
MOV(021) #0 Actv_M

## Function block Shift_Ary
VAR_INPUT
  Fst_indx : INT;
  Lst_indx : INT;
  cmd : BOOL;
END_VAR
VAR_IN_OUT
  Ary : ARRAY[0..99] OF INT;
END_VAR
VAR
  itr : INT;
  nxt_itr : INT;
END_VAR
IF cmd THEN
	
FOR itr := Fst_indx TO Lst_indx-1 DO
	nxt_itr := itr+1;
Ary[itr] := Ary[nxt_itr];
END_FOR;

Ary[Lst_indx] := 0;

END_IF;